Fanuc KAREL source: kt00567.KL

-- PROVISIONAL review KL for V770-1; original PC SHA256 f2c30c87b8c486beeec19175d4488633ffb376dbfcdc331f73e700d7b422d3db
-- Incomplete behavior may be omitted. Consult companion uncertainty JSON. Do not deploy.
PROGRAM KT00567
%NOLOCKGROUP
VAR
  R2 : REAL
-- UNRESOLVED_DECL V1 type=000013
-- UNRESOLVED_DECL OUT type=000013
BEGIN
  -- UNRESOLVED_PC offsets 5-20; opcodes 2E,22,32,35
  -- UNRESOLVED_PC offsets 25-36; opcodes 2E,23
  -- UNRESOLVED_PC offsets 41-63; opcodes 49,21,8A,4A
  -- UNRESOLVED_PC offsets 68-72; opcodes 7F
END KT00567
